// Mitsubishi GX Works2 project: 7   PLC: FX2N/FX2NC

PROGRAM MAIN
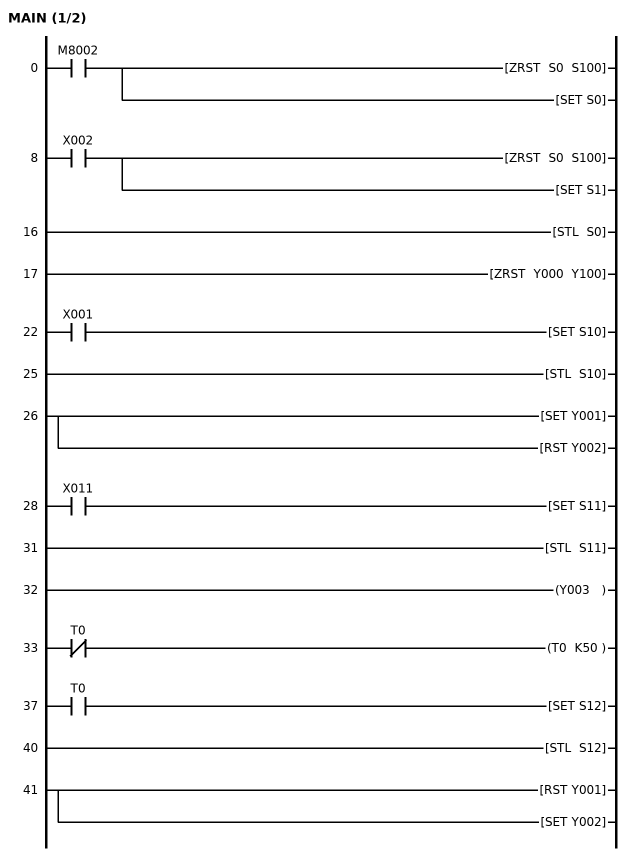
0     LD      M8002
      ZRST    S0 S100
      SET     S0
8     LD      X002
      ZRST    S0 S100
      SET     S1
16    STL     S0
17    ZRST    Y000 Y100
22    LD      X001
      SET     S10
25    STL     S10
26    SET     Y001
      RST     Y002
28    LD      X011
      SET     S11
31    STL     S11
32    OUT     Y003
33    LDI     T0
      OUT     T0 K50
37    LD      T0
      SET     S12
40    STL     S12
41    RST     Y001
      SET     Y002
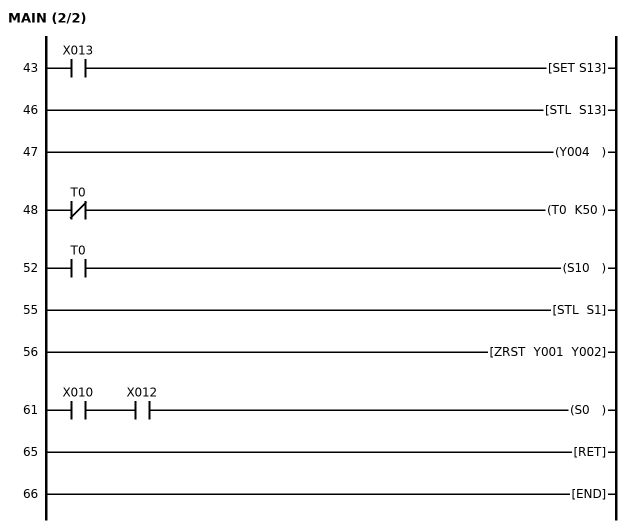
43    LD      X013
      SET     S13
46    STL     S13
47    OUT     Y004
48    LDI     T0
      OUT     T0 K50
52    LD      T0
      OUT     S10
55    STL     S1
56    ZRST    Y001 Y002
61    LD      X010
      AND     X012
      OUT     S0
65    RET
66    END
END_PROGRAM

// device comments not shown above
BL0  ; main
BL1  ; a
BL2  ; b
